{attribute 'no_check'}
//Default IOs of a Publisher network variable 
FUNCTION_BLOCK EAP_PUB_VAR 
VAR_OUTPUT CONSTANT
END_VAR
VAR_INPUT
	VarId						AT %Q*:	UINT;
	{attribute 'displaymode':='hex'}
	VarCtrl						AT %Q*:	UINT;
END_VAR		
VAR_OUTPUT	
	{attribute 'displaymode':='hex'}
	VarState					AT %I*:	UINT;
	
	NotSentVarSkipped					:	BOOL;
END_VAR
VAR
END_VAR

	(* IOs 									*)
	(****************************************)

NotSentVarSkipped							:= VarState.0;

PROPERTY PUBLIC disablePublishing : BOOL
GET
disablePublishing		:= VarCtrl.0;
END_GET
SET
VarCtrl.0				:= disablePublishing;
END_SET
END_PROPERTY

END_FUNCTION_BLOCK

(* stored: Version 1.1.0.1, ProductVersion 3.1.4024.13
   POU EAP_PUB_VAR: Id {04dd49ad-caf7-4506-9575-9e5dd17759ca}, SpecialFunc None
   Property disablePublishing: Id {f4b8d7e0-0241-483a-a4a4-479c23d84699}
   Get Get: Id {9c3f7f8a-66aa-4dea-a347-fd719c92840e}
   Set Set: Id {1add8aae-11f4-4ca8-93d2-72e497741520} *)
